//{attribute 'qualified_only'}
//{attribute 'strict'}
TYPE E_TORQUE_Scaling : (
	//E_TORQUE_IDLE,
	//E_TORQUE_GETPORTNO,
	//E_TORQUE_RATEDCURRENT,
	//E_TORQUE_MAXCURRENT,
	//E_TORQUE_MONITOR,
	//E_TORQUE_ERROR,
	E_TORQUE_DUMMY
);
END_TYPE

(* stored: Version 1.1.0.1
   DUT E_TORQUE_Scaling: Id {a1a6e498-de91-4abe-88f3-81147e8fa1f4} *)
